TYPE E_MachineMode :
(
	auto,
	manual,
	none
);
END_TYPE

(* stored: Version 1.1.0.1, ProductVersion 3.1.4024.16
   DUT E_MachineMode: Id {98f966c2-e918-4fda-87f0-3893ed20f891} *)
